TYPE ChamberConfigs :
STRUCT
	PsdChamberConfig : PsdChamberConfig;
	LightspeedChamberConfig : LightspeedChamberConfig;	
	PhotoLumChamberConfig : PhotoLumChamberConfig;
END_STRUCT
END_TYPE

(* stored: Version 1.1.0.1, ProductVersion 3.1.4024.12
   DUT ChamberConfigs: Id {070692ba-a1e1-401c-ac7d-6be18ed0dc4c} *)
